SUBAPPLICATION mapping_OUTPUT (* Subapplication Type *)
  (* Standard: 61499-2 *)
  (* Version 1.0, 2023-02-07, franz *)
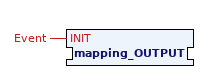
  EVENT_INPUT
    INIT;
  END_EVENT
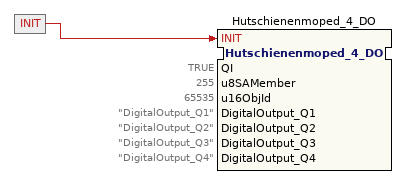
  FBS
    Hutschienenmoped_4_DO : Hutschienenmoped_4_DO(QI := TRUE, u8SAMember := 255, u16ObjId := 65535, DigitalOutput_Q1 := "DigitalOutput_Q1", DigitalOutput_Q2 := "DigitalOutput_Q2", DigitalOutput_Q3 := "DigitalOutput_Q3", DigitalOutput_Q4 := "DigitalOutput_Q4");
  END_FBS
  EVENT_CONNECTIONS
    INIT TO Hutschienenmoped_4_DO.INIT;
  END_CONNECTIONS
END_SUBAPPLICATION
